# B&R Automation Studio project proyecto_dardos
Automation Studio 4.9

## Configuration Config1

CPU 4PPC70.0702-23B, AutomationRuntime B4.92, Build 4.1.2, Vc V4.72.5

### Task classes (Cpu.sw)
```
Cyclic#1:
  dardos <- Libraries.dardos.dardos.prg
Cyclic#4:
  Program1 <- radios.Program.prg
VcDataObjects: Visu_d <- Libraries.dardos.Visu_dardos.dob
Binaries: vcctext, arialbd, vccpiech, vcmgr, vccpopup, Visu_d02, vcxml, vccdt, vccshape, Visu_d03, vcchspot, vcnet, vcdsloc, vcbclass, vcfntttf, vcdsint, vctcal, vcshared, vcrt, vcpk, vccbmp, TCData, vcfile, vccbtn, vccslider, vccddbox, vcptelo, vcalarm, vcpdi855, Visu_d01, vccnum, vcpdsw, FWRules, vccdbox, arial, vccovl, visvc, udbdef, vccscale, vccline, vcpdvnc, vcpfar00, vccalarm, vccstr, vcchtml, vcpdi815, vcpfppc7, vcctrend, vcgclass, vcclbox, vccurl, vcpdihd, Role, arconfig, User, asfw, ashwd, ashwac, sysconf, iomap
Libraries: visapi, asieccon, fileio, dataobj, vcresman, runtime, astime
```

### Hardware
```
4PPC70_0702_23B : 4PPC70.0702-23B v1.5.4.0
  Connector IF2:
    ActivateDevice = 1
  ConfigurationID = juego_dardos_Config1
  Simulation = 1
  FileDevice1
  FileDeviceName1 = USER
  FileDevicePath1 = USER_PATH
  VcObjectName = Visu_d
  KeyMappingFile = VC\4PPC70_0702_23B.dis
```

## Logical view

Binary libraries used (declarations not repeated): operator, runtime, astime, AsIecCon, visapi

### Global.typ - Global data types
```iecst
TYPE
	gmain_enum :
		(
		etapa_2,
		etapa_1
		);
END_TYPE
```

### Global.var - Global variables
```iecst
VAR
	radio : UINT;
	y_posicion : UDINT;
	x_posicion : UDINT;
	current_page : USINT;
	VC_HANDLE : UDINT;
	touch_status : UDINT;
	touch : TouchAction;
	ready : BOOL;
	ancho_alto : ARRAY[1..7] OF UINT;
	circulo : USINT;
	touch_real : REAL;
	touch_active : BOOL;
	diametro_touch : REAL;
	estado : gmain_enum;
END_VAR
VAR CONSTANT
	y : UINT := 230;
	x : UINT := 230;
END_VAR
VAR
	x_real : REAL;
	y_real : REAL;
	x_posicion_real : REAL;
	y_posicion_real : REAL;
	puntaje_acumulado : UINT;
	update_puntaje : BOOL;
	updateRadio : BOOL;
	valor_score : UINT;
	cantidad_tiros : USINT;
	puntaje_intermediario : ARRAY[1..7] OF UINT;
	puntaje : UINT;
	segment_score : UINT;
END_VAR
```

### Package Logical/Libraries - Global libraries

### Program Logical/Libraries/dardos/dardos (IEC)

#### Main.st - Init, cyclic, exit code
```iecst
PROGRAM _INIT
	(* Insert code here *)
	listo := 0;
	VC_HANDLE := 0;
//	x := 230;
//	y := 230;
	relleno := 250;
	perimetro_color := 0;
	ready := 0;
	ancho_alto;
	circulo := 0;

	x_posicion;
	y_posicion;

	ancho_alto [7] := 350;
	ancho_alto [6] := 300;
	ancho_alto [5] := 250;
	ancho_alto [4] := 200;
	ancho_alto [3] := 150;
	ancho_alto [2] := 100;
	ancho_alto [1] := 50;

	fill [7] := 164;
	fill [6] := 250;
	fill [5] := 164;
	fill [4] := 250;
	fill [3] := 164;
	fill [2] := 250;
	fill [1] := 19;

END_PROGRAM

PROGRAM _CYCLIC
	(* Insert code here *)

	touch;
	current_page;

// habilitar variable con teclado //

	IF updateRadio THEN
		VA_Redraw (1,VC_HANDLE);
	END_IF;
	// habilitar setup //
	VC_HANDLE := VA_Setup(1,SPD);
	IF VC_HANDLE <> 0 THEN
		ready := 1;

		ELSE VC_HANDLE := 0;
	END_IF;
	// empezar a dibujar //

//	IF ready = 1 AND current_page = 18 THEN
//		IF VA_Saccess(1,VC_HANDLE) = 0  THEN
//			VA_Rect(1,VC_HANDLE,50,50,400,360,250,0);
//			VA_Ellipse (1,VC_HANDLE,x,y,ancho_alto,ancho_alto,color,0);
//		END_IF;
//		END_IF;
	//dibujo en estado inicial //
	IF ready = 1 AND current_page = 18  THEN
		IF VA_Saccess(1,VC_HANDLE) = 0  THEN
			VA_GetTouchAction (1,VC_HANDLE,1,ADR(touch));
			x_posicion := touch.x;
			y_posicion := touch.y;
			touch_status := touch.status;
			VA_Rect(1,VC_HANDLE,50,50,370,360,11,0);
    		VA_Ellipse (1,VC_HANDLE,x,y,ancho_alto[7],ancho_alto[7],fill[7],0);
			VA_Ellipse (1,VC_HANDLE,x,y,ancho_alto[6],ancho_alto[6],fill[6],0);
			VA_Ellipse (1,VC_HANDLE,x,y,ancho_alto[5],ancho_alto[5],fill[5],0);
			VA_Ellipse (1,VC_HANDLE,x,y,ancho_alto[4],ancho_alto[4],fill[4],0);
			VA_Ellipse (1,VC_HANDLE,x,y,ancho_alto[3],ancho_alto[3],fill[3],0);
			VA_Ellipse (1,VC_HANDLE,x,y,ancho_alto[2],ancho_alto[2],fill[2],0);
			VA_Ellipse (1,VC_HANDLE,x,y,ancho_alto[1],ancho_alto[1],fill[1],0);
			VA_Srelease (1,VC_HANDLE);
		END_IF;
	END_IF;

	//los posibles circulos y sus tamaños//

	IF circulo = 7 AND updateRadio THEN

			updateRadio := FALSE;
			ancho_alto[7] := radio;
		    fill[7] := 164;
	END_IF;

	IF circulo = 6 AND updateRadio THEN
		updateRadio := FALSE;

			ancho_alto[6] := radio;
			fill [6] := 250;
		END_IF;

		IF circulo = 5 AND updateRadio THEN
			updateRadio := FALSE;

		ancho_alto[5] := radio;
		fill [5] := 164;

	END_IF;

		IF circulo = 4 AND updateRadio THEN
		updateRadio := FALSE;

		ancho_alto[4] := radio;
		fill [4] := 250;

	END_IF;

		IF circulo = 3 AND updateRadio THEN
		updateRadio := FALSE;

		ancho_alto[3] := radio;
		fill [3] := 164;

			END_IF;

		IF circulo = 2 AND updateRadio THEN
		updateRadio := FALSE;

		ancho_alto[2] := radio;
		fill [2] := 250;

		END_IF;

    	IF circulo = 1 AND updateRadio THEN
		updateRadio := FALSE;

		ancho_alto[1] := radio;
		fill [1] := 19;

	END_IF;

END_PROGRAM

PROGRAM _EXIT
	(* Insert code here *)

END_PROGRAM
```

#### Variables.var - Local variables
```iecst
VAR
	listo : UINT;
	relleno : UINT;
	perimetro_color : UINT;
	SPD : STRING[80] := 'Visu_d';
	status_attach : UINT;
	variable_1 : UINT;
	variable_2 : UINT;
	variable_3 : UINT;
	variable_4 : UINT;
	variable_5 : UINT;
	variable_6 : UINT;
	variable_7 : UINT;
	xrect : UINT;
	yrec : UINT;
	widthrect : UINT;
	heithRect : UINT;
	colorRec : USINT;
	fillRec : USINT;
	fill : ARRAY[1..7] OF UINT;
END_VAR
```

- Visualisation Logical/Libraries/dardos/Visu_dardos (not shown)

### Program Logical/radios/Program

#### Variables.var
```iecst
VAR
	resetear : BOOL;
END_VAR
```

#### Main.st
```iecst
PROGRAM _INIT
	(* Insert code here *)
	puntaje_intermediario[7] := 70;
	puntaje_intermediario[6] := 60;
	puntaje_intermediario[5] := 50;
	puntaje_intermediario[4] := 40;
	puntaje_intermediario[3] := 30;
	puntaje_intermediario[2] := 20;
	puntaje_intermediario[1] := 10;
END_PROGRAM

PROGRAM _CYCLIC
	// VALOR DEL DIAMETRO EN CUALQUIER PUNTO DE LA PANTALLA PARA TOMAR VALORES ENTRE LOS CIRCULOS //
	x_real := UINT_TO_REAL (x);
	y_real := UINT_TO_REAL (y);
	x_posicion_real := UDINT_TO_REAL (x_posicion);
	y_posicion_real := UDINT_TO_REAL (y_posicion);
diametro_touch := (SQRT ((EXPT((x_real-x_posicion_real),2)) + (EXPT((y_real-y_posicion_real),2))))*2;
//VALOR DE LOS PUNTAJES//

	IF  diametro_touch < ancho_alto[7] AND diametro_touch >= ancho_alto[6] THEN
		IF current_page = 18 AND EDGEPOS (touch_status = 1) THEN
			valor_score := puntaje_intermediario[7];
			ELSE valor_score := 0;
		END_IF;
			END_IF;

	IF diametro_touch < ancho_alto [6] AND diametro_touch >= ancho_alto [5] THEN
			IF current_page = 18 AND EDGEPOS (touch_status = 1) THEN
				valor_score := puntaje_intermediario [6];
			ELSE valor_score := 0;
			END_IF;
		END_IF;

	IF diametro_touch < ancho_alto [5] AND diametro_touch >= ancho_alto [4] THEN
		IF current_page = 18 AND EDGEPOS (touch_status = 1) THEN
			valor_score := puntaje_intermediario [5];
		ELSE valor_score := 0;
		END_IF;
	END_IF;

	IF diametro_touch < ancho_alto [4] AND diametro_touch >= ancho_alto [3] THEN
		IF current_page = 18 AND EDGEPOS (touch_status = 1) THEN
			valor_score := puntaje_intermediario [4];
		ELSE valor_score := 0;
		END_IF;
	END_IF;

	IF diametro_touch < ancho_alto [3] AND diametro_touch >= ancho_alto [2] THEN
		IF current_page = 18 AND EDGEPOS (touch_status = 1) THEN
			valor_score := puntaje_intermediario [3];
				ELSE valor_score := 0;
		END_IF;
	END_IF;

	IF diametro_touch < ancho_alto [2] AND diametro_touch >= ancho_alto [1] THEN
		IF current_page = 18 AND EDGEPOS (touch_status = 1) THEN
			valor_score := puntaje_intermediario [2];
				ELSE valor_score := 0;
		END_IF;
	END_IF;

	IF diametro_touch < ancho_alto [1]  THEN
		IF current_page = 18 AND EDGEPOS (touch_status = 1) THEN
			valor_score := puntaje_intermediario[1];
				ELSE valor_score := 0;
		END_IF;
	END_IF;

	//elegir los puntajes para cada circulo //

	IF segment_score = 7 AND update_puntaje THEN
		update_puntaje := FALSE;
		puntaje_intermediario [7] := puntaje;
	END_IF;

	IF segment_score = 6 AND update_puntaje THEN
		update_puntaje := FALSE;
		puntaje_intermediario [6] := puntaje;
	END_IF;

	IF segment_score = 5 AND update_puntaje THEN
		update_puntaje := FALSE;
		puntaje_intermediario [5] := puntaje;
	END_IF;

	IF segment_score = 4 AND update_puntaje THEN
		update_puntaje := FALSE;
		puntaje_intermediario [4] := puntaje;
	END_IF;

	IF segment_score = 3 AND update_puntaje THEN
		update_puntaje := FALSE;
		puntaje_intermediario [3] := puntaje;
	END_IF;

	IF segment_score = 2 AND update_puntaje THEN
		update_puntaje := FALSE;
		puntaje_intermediario [2] := puntaje;
	END_IF;

	IF segment_score = 1 AND update_puntaje THEN
		update_puntaje := FALSE;
		puntaje_intermediario [1] := puntaje;
	END_IF;

	// valor de puntaje acumulado //
	puntaje_acumulado := puntaje_acumulado + valor_score;

	//cantidad de tiros //
	IF current_page = 18 AND EDGEPOS (touch_status =1) AND resetear = FALSE AND x_posicion > 50 AND x_posicion < 420 AND y_posicion > 50 AND y_posicion < 410 THEN
	  cantidad_tiros := cantidad_tiros +1;
	END_IF;

	//resetear puntos y tiros //

	IF EDGEPOS (resetear)  THEN
		cantidad_tiros := 0;
		puntaje_acumulado := 0;
		ELSE resetear := FALSE;

	END_IF;

END_PROGRAM

PROGRAM _EXIT
	(* Insert code here *)

END_PROGRAM
```

Listed in the project but not available here: Logical/Libraries/dardos/dardos/Types.typ
